# EPICS substitutions: fgccmdSup/Db/fgccmd_test.substitutions
# ../../sw/kt/fgcepics/fgccmdSup/Db/fgccmd_class_63.substitutions - This file is automatically generated by `parser/Output/EPICS/records/cmd_records.pm`

# This is a template file - RECORD names can be edited!

##########################################
# Command/response records for class 63  #
##########################################

# Note (!):
# SET records: ':S' will be appended to record name
# GET records: ':G' will be appended to record name

######## Long string properties (decoded bitmask) ########

file "fgccmd_w_string_get.template"
{
pattern
{ RECORD          , PROP        , NELM , DESC }
{ "STATUS:FAULTS" , "FGC.FAULTS", 256  , ""   }
}

file "fgccmd_w_string_set.template"
{
pattern
{ RECORD          , PROP        , NELM , DESC }
}

######## String properties (decoded enum) ########

file "fgccmd_string_get.template"
{
pattern
{ RECORD     , PROP       , DESC }
{ "TEST:CHAR", "TEST.CHAR", ""   }
}

file "fgccmd_string_set.template"
{
pattern
{ RECORD , PROP , DESC }
{ "TEST:CHAR", "TEST.CHAR", ""   }
}

######## Real type properties ########

file "fgccmd_real_get.template"
{
pattern
{ RECORD         , PROP         , EGU , PREC , DESC }
{ "TEST:FLOAT"   , "TEST.FLOAT" , ""  , "6"  , ""   }
}

file "fgccmd_real_set.template"
{
pattern
{ RECORD         , PROP         , EGU , PREC , DESC }
{ "TEST:FLOAT"   , "TEST.FLOAT" , ""  , "6"  , ""   }
}

######## Long type properties ########

file "fgccmd_long_get.template"
{
pattern
{ RECORD          , PROP          , EGU     , DESC                          }
{ "TEST:INT16S"   , "TEST.INT16S" , ""      , ""                            }
{ "TEST:INT16U"   , "TEST.INT16U" , ""      , ""                            }
{ "TEST:INT32S"   , "TEST.INT32S" , ""      , ""                            }
{ "TEST:INT32U"   , "TEST.INT32U" , ""      , ""                            }
{ "TEST:INT8S"    , "TEST.INT8S"  , ""      , ""                            }
{ "TEST:INT8U"    , "TEST.INT8U"  , ""      , ""                            }
}

file "fgccmd_long_set.template"
{
pattern
{ RECORD          , PROP          , EGU     , DESC                          }
{ "TEST:INT16S"   , "TEST.INT16S" , ""      , ""                            }
{ "TEST:INT16U"   , "TEST.INT16U" , ""      , ""                            }
{ "TEST:INT32S"   , "TEST.INT32S" , ""      , ""                            }
{ "TEST:INT32U"   , "TEST.INT32U" , ""      , ""                            }
{ "TEST:INT8S"    , "TEST.INT8S"  , ""      , ""                            }
{ "TEST:INT8U"    , "TEST.INT8U"  , ""      , ""                            }
}

######## Reference table properties (TIME,REF) ########

file "fgccmd_table_arr.template"
{
pattern
{ RECORD , PROP , NELM_DOUBLE , PREC, DESC }
}

file "fgccmd_table_get.template"
{
pattern
{ RECORD , PROP , NELM_DOUBLE , NELM_CHAR , TIME_ARRAY , REF_ARRAY, DESC }
}

file "fgccmd_table_set.template"
{
pattern
{ RECORD , PROP , NELM_DOUBLE , NELM_CHAR , TIME_ARRAY , REF_ARRAY , DESC }
}

# End of file: ../../sw/kt/fgcepics/fgccmdSup/Db/fgccmd_class_63.substitutions
